// TIA Portal V20 export
FUNCTION "03 T1-A ARUNC Aux" : Void   // FC1302, LAD
TITLE = AUXILIARIES
{ S7_Optimized_Access := 'TRUE' }
// stored: AutoNumber false, SetENOAutomatically false
   VAR_TEMP
      Aux_OS : Bool;
      Aux_sup : Real;
      Aux_inf : Real;
      Aux_DInt : DInt;
      Aux_Real : Real;
   END_VAR
   VAR CONSTANT
      "Max differenza L tubi" : Real := 500.0;
   END_VAR
   VAR_TEMP   // added for the SCL form of the ladder/FBD networks
      _w1 : Bool;
      _w2 : Bool;
   END_VAR
BEGIN

REGION Network 1: =========== MEMORIES ===========
END_REGION

REGION Network 2: Piece presence
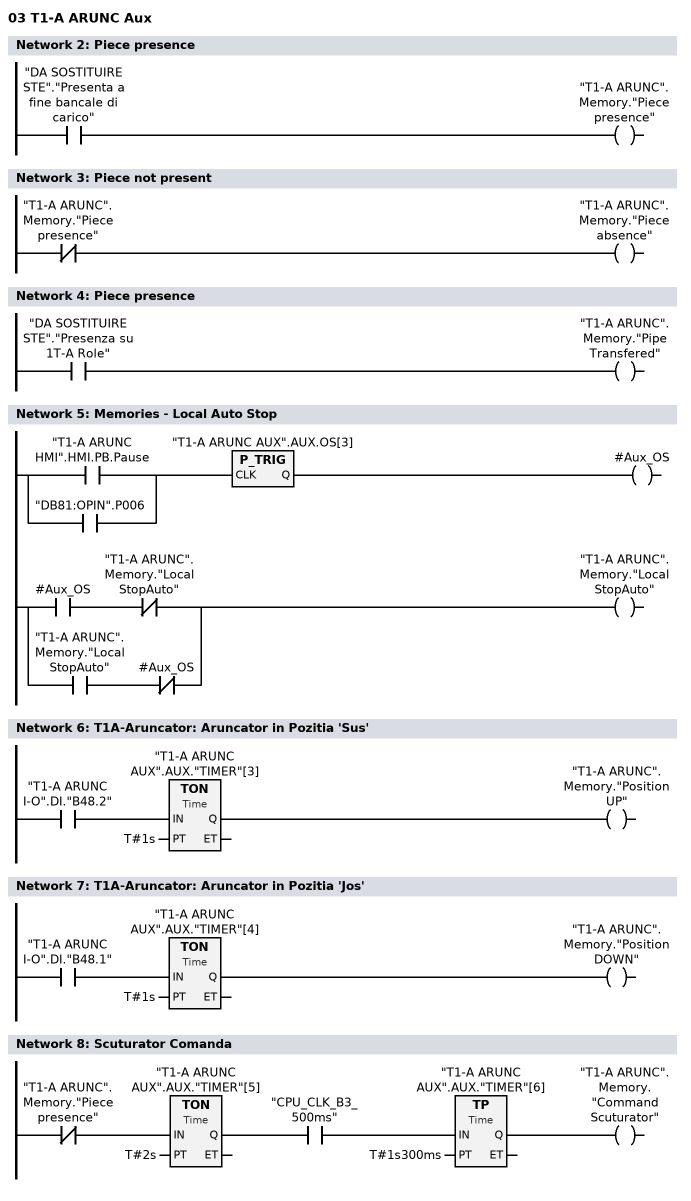
   RUNG wire#powerrail
      Contact( "DA SOSTITUIRE STE"."Presenta a fine bancale di carico" )
      Coil( "T1-A ARUNC".Memory."Piece presence" )
   END_RUNG
   // the same network as SCL:
   "T1-A ARUNC".Memory."Piece presence" := "DA SOSTITUIRE STE"."Presenta a fine bancale di carico";
END_REGION

REGION Network 3: Piece not present
   RUNG wire#powerrail
      I_Contact( "T1-A ARUNC".Memory."Piece presence" )
      Coil( "T1-A ARUNC".Memory."Piece absence" )
   END_RUNG
   // the same network as SCL:
   "T1-A ARUNC".Memory."Piece absence" := NOT "T1-A ARUNC".Memory."Piece presence";
END_REGION

REGION Network 4: Piece presence
   RUNG wire#powerrail
      Contact( "DA SOSTITUIRE STE"."Presenza su 1T-A Role" )
      Coil( "T1-A ARUNC".Memory."Pipe Transfered" )
   END_RUNG
   // the same network as SCL:
   "T1-A ARUNC".Memory."Pipe Transfered" := "DA SOSTITUIRE STE"."Presenza su 1T-A Role";
END_REGION

REGION Network 5: Memories - Local Auto Stop
   RUNG wire#powerrail
      Contact( "T1-A ARUNC HMI".HMI.PB.Pause )
      wire#w1
      P_Trig( "T1-A ARUNC AUX".AUX.OS[3] )
      Coil( #Aux_OS )
   END_RUNG
   RUNG wire#powerrail
      Contact( "DB81:OPIN".P006 )
   END_RUNG wire#w1
   RUNG wire#powerrail
      Contact( #Aux_OS )
      I_Contact( "T1-A ARUNC".Memory."Local StopAuto" )
      wire#w2
      Coil( "T1-A ARUNC".Memory."Local StopAuto" )
   END_RUNG
   RUNG wire#powerrail
      Contact( "T1-A ARUNC".Memory."Local StopAuto" )
      I_Contact( #Aux_OS )
   END_RUNG wire#w2
   // the same network as SCL:
   #_w1 := "T1-A ARUNC HMI".HMI.PB.Pause OR "DB81:OPIN".P006;
   #_w2 := #_w1 AND NOT "T1-A ARUNC AUX".AUX.OS[3];   // rising edge
   "T1-A ARUNC AUX".AUX.OS[3] := #_w1;
   #Aux_OS := #_w2;
   "T1-A ARUNC".Memory."Local StopAuto" := (#Aux_OS AND NOT "T1-A ARUNC".Memory."Local StopAuto") OR ("T1-A ARUNC".Memory."Local StopAuto" AND NOT #Aux_OS);
END_REGION

REGION Network 6: T1A-Aruncator: Aruncator in Pozitia 'Sus'
   RUNG wire#powerrail
      Contact( "T1-A ARUNC I-O".DI."B48.2" )
      { S7_Templates := "time_type := Time" } "T1-A ARUNC AUX".AUX."TIMER"[3].TON(pt := T#1s, et =>)
      Coil( "T1-A ARUNC".Memory."Position UP" )
   END_RUNG
   // the same network as SCL:
   "T1-A ARUNC AUX".AUX."TIMER"[3].TON(IN := "T1-A ARUNC I-O".DI."B48.2", PT := T#1s);
   "T1-A ARUNC".Memory."Position UP" := "T1-A ARUNC AUX".AUX."TIMER"[3].Q;
END_REGION

REGION Network 7: T1A-Aruncator: Aruncator in Pozitia 'Jos'
   RUNG wire#powerrail
      Contact( "T1-A ARUNC I-O".DI."B48.1" )
      { S7_Templates := "time_type := Time" } "T1-A ARUNC AUX".AUX."TIMER"[4].TON(pt := T#1s, et =>)
      Coil( "T1-A ARUNC".Memory."Position DOWN" )
   END_RUNG
   // the same network as SCL:
   "T1-A ARUNC AUX".AUX."TIMER"[4].TON(IN := "T1-A ARUNC I-O".DI."B48.1", PT := T#1s);
   "T1-A ARUNC".Memory."Position DOWN" := "T1-A ARUNC AUX".AUX."TIMER"[4].Q;
END_REGION

REGION Network 8: Scuturator Comanda
   RUNG wire#powerrail
      I_Contact( "T1-A ARUNC".Memory."Piece presence" )
      { S7_Templates := "time_type := Time" } "T1-A ARUNC AUX".AUX."TIMER"[5].TON(pt := T#2s, et =>)
      Contact( "CPU_CLK_B3_500ms" )
      { S7_Templates := "time_type := Time" } "T1-A ARUNC AUX".AUX."TIMER"[6].TP(pt := T#1s300ms, et =>)
      Coil( "T1-A ARUNC".Memory."Command Scuturator" )
   END_RUNG
   // the same network as SCL:
   "T1-A ARUNC AUX".AUX."TIMER"[5].TON(IN := NOT "T1-A ARUNC".Memory."Piece presence", PT := T#2s);
   "T1-A ARUNC AUX".AUX."TIMER"[6].TP(IN := "T1-A ARUNC AUX".AUX."TIMER"[5].Q AND "CPU_CLK_B3_500ms",
                           PT := T#1s300ms);
   "T1-A ARUNC".Memory."Command Scuturator" := "T1-A ARUNC AUX".AUX."TIMER"[6].Q;
END_REGION
END_FUNCTION
